// TIA Portal V17 export
// export: Created 2022-07-04T12:17:16.4924558Z, ExportSetting WithDefaults, DisplayName Totally Integrated Automation Portal, DisplayVersion V17, DisplayName TIA Portal Openness, DisplayVersion V17, DisplayName TIA Portal Version Control Interface, DisplayVersion V17, DisplayName STEP 7 Professional, DisplayVersion V17, DisplayName STEP 7 Safety, DisplayVersion V17, DisplayName WinCC Advanced, DisplayVersion V17
ORGANIZATION_BLOCK "Main"   // OB1, LAD, ProgramCycle
TITLE = "Main Program Sweep (Cycle)"
{ S7_Optimized_Access := 'TRUE' }
VERSION : 0.1
// stored: AutoNumber true, IsIECCheckEnabled false, SetENOAutomatically false
   VAR_INPUT
      Initial_Call : Bool;   // Initial call of this OB
      Remanence : Bool;   // =True, if remanent data are available
   END_VAR
BEGIN

REGION Network 1
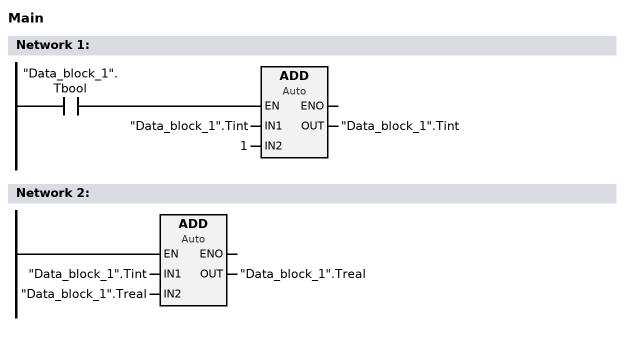
   RUNG wire#powerrail
      Contact( "Data_block_1".Tbool )
      Add(in1 := "Data_block_1".Tint, in2 := 1, out => "Data_block_1".Tint)
   END_RUNG
   // the same network as SCL:
   IF "Data_block_1".Tbool THEN "Data_block_1".Tint := "Data_block_1".Tint + 1; END_IF;
END_REGION

REGION Network 2
   RUNG wire#powerrail
      Add(in1 := "Data_block_1".Tint, in2 := "Data_block_1".Treal, out => "Data_block_1".Treal)
   END_RUNG
   // the same network as SCL:
   "Data_block_1".Treal := "Data_block_1".Tint + "Data_block_1".Treal;
END_REGION
END_ORGANIZATION_BLOCK
